// TwinCAT 3 PLC project TcSocketHelper_SingleServerBinary
// ProgramVersion: 3.1.0.5
// libraries:
//   Tc2_Standard, * (Beckhoff Automation GmbH)
//   Tc2_System, * (Beckhoff Automation GmbH)
//   Tc2_TcpIp, * (Beckhoff Automation GmbH)
//   Tc2_Utilities, * (Beckhoff Automation GmbH)
//   Tc3_Module, * (Beckhoff Automation GmbH)
// project tree:
//   Data types/ ST_ApplicationBinaryData.TcDUT, ST_BinaryFrame.TcDUT, ST_BinaryHeader.TcDUT
//   Global Variables/ Global_Variables.TcGVL
//   / PlcTaskServer.TcTTO
//   POUs/ FB_Server.TcPOU, FB_ServerApplication.TcPOU, FB_ServerConnection.TcPOU, MAIN.TcPOU
//   POUs/Helper POUs/ FB_FrameFifo.TcPOU (not stored), FB_LogFifo.TcPOU, F_ADSLOGHEXDATA.TcPOU
// real-time tasks:
//   TASK PlcTaskServer: cycle T#10ms, priority 21, ADS port 351

CONFIGURATION TcSocketHelper_SingleServerBinary
    RESOURCE PLC ON TwinCAT3
        TASK PlcTaskServer(INTERVAL := T#10ms, PRIORITY := 21);
        PROGRAM MAIN WITH PlcTaskServer : MAIN;
    END_RESOURCE
END_CONFIGURATION

// ---- Data types/ST_ApplicationBinaryData.TcDUT
(* Simple binary user data (8 byte aligned) *)
TYPE ST_ApplicationBinaryData :
STRUCT
	(* Adapt this structure to match your protocol needs *)
	
	dtTimeStamp : DT		:= DT#2008-12-01-00:00;(* 4 byte *)
	nVelo		: UDINT		:= 0;(* 4 byte *)
	fPos		: LREAL		:= 0.0;(* 8 byte *)
	arr	 		: ARRAY[0..19] OF BYTE;(* 20 byte *)

	sMsg		: STRING	:= 'None';(* 81 byte *)
	reserved	: ARRAY[0..2] OF BYTE;(* Alignment data: 3 byte *)

	(* Total user data size = 120 byte *)
END_STRUCT
END_TYPE

// ---- Data types/ST_BinaryFrame.TcDUT
(* Simple binary TCP/IP frame (8 byte aligned) *)
TYPE ST_BinaryFrame :
STRUCT
	head	: ST_BinaryHeader;(* Frame header (16 byte) *)
	data 	: ST_ApplicationBinaryData;(* User data (120 byte) *)

	(* Total frame size = 136 byte *)
END_STRUCT
END_TYPE

// ---- Data types/ST_BinaryHeader.TcDUT
(* Simple binary TCP/IP frame header (8 byte aligned) *)
TYPE ST_BinaryHeader :
STRUCT
	dwStart		: DWORD	:= 16#BECF1234;	(* Start bytes *)
	cbLength	: UDINT(0..PLCPRJ_BUFFER_SIZE) := 0;(* Max. length of attached binary data *)
	nS			: UDINT := 0;(* Send counter *)
	nR			: UDINT	:= 0;(* Receive counter *)
	
	(* Total header data size = 16 byte *)
END_STRUCT
END_TYPE

// ---- Global Variables/Global_Variables.TcGVL
VAR_GLOBAL CONSTANT
	PLCPRJ_BUFFER_SIZE						: UDINT := 1000;(* Max. internal fifo/receiver buffer size *)

(*	PLCPRJ_CLIENT_SEND_CYCLE_TIME			: TIME := T#1S; not used at server side *)
	PLCPRJ_RECEIVE_POLLING_TIME				: TIME := T#100MS;
	PLCPRJ_RECEIVE_TIMEOUT					: TIME := T#50S;

	(* Some project specific error codes *)
	PLCPRJ_ERROR_RECEIVE_TIMEOUT			: UDINT := 16#8101;(* Receive timeout *)
	PLCPRJ_ERROR_SENDFIFO_OVERFLOW			: UDINT := 16#8102;(* Send fifo overflow *)
	PLCPRJ_ERROR_RECFIFO_OVERFLOW			: UDINT := 16#8103;(* Receive fifo overflow *)
	PLCPRJ_ERROR_INVALID_FRAME_FORMAT		: UDINT := 16#8104;(* Invalid frame format/data *)
END_VAR

// ---- POUs/MAIN.TcPOU
PROGRAM MAIN
VAR
	sSrvNetID		: T_AmsNetID	:= '';(* TwinCAT TCP/IP server network address *)
	sLocalHost		: T_Ipv4Addr 	:= '127.0.0.1';(* Server IP network address *)
	nLocalPort		: UDINT 		:= 200;(* Server port number *)
	bEnable			: BOOL 			:= TRUE;(* TRUE => Enable server data exchange, FALSE => Disable *)
	bLog			: BOOL			:= TRUE;(* TRUE => Enable log message output, FALSE => Disable *)
	fbServer		: FB_Server := ( sPrefix := 'SERVER::' );(* Server (connection) instance *)
	hServer			: T_HSERVER;(* Server connection handle *)

	fbCloseAll		: FB_SocketCloseAll;
	bInitialize		: BOOL := TRUE;
END_VAR

(* On PLC reset or program download close all old (opened) connections *)
fbCloseAll( sSrvNetID := sSrvNetID, bExecute:= bInitialize );
IF fbCloseAll.bBusy OR fbCloseAll.bError THEN
	RETURN;
END_IF

IF bInitialize THEN
	bInitialize := FALSE;

	(* Initialize server handle *)
	F_CreateServerHnd( 	sSrvNetID 	:= sSrvNetID,
						sLocalHost 	:= sLocalHost,
						nLocalPort	:= nLocalPort,
						nMode 		:= SEL( bLog, 0, CONNECT_MODE_ENABLEDBG ),(* Enable debug messages *)
						bEnable 	:= FALSE,(* TRUE = leave listener socket open, FALSE = close listener socket after last connection ist closed too *)
						hServer 	:= hServer );
END_IF


(* Trigger the execution of every server (connection) instance *)
fbServer( hServer := hServer, sSrvNetID := sSrvNetID, bEnable := bEnable, bLog := bLog );

END_PROGRAM

// ---- POUs/FB_Server.TcPOU
FUNCTION_BLOCK FB_Server
VAR_IN_OUT
	hServer			: T_HSERVER;(* Server connection handle *)
END_VAR
VAR_INPUT
	sSrvNetID		: T_AmsNetID	:= '';(* TwinCAT TCP/IP server network address *)
	bEnable			: BOOL 			:= FALSE;(* TRUE => Enable server data exchange, FALSE => Disable *)
	bLog			: BOOL 			:= FALSE;(* TRUE => Enable log message output, FALSE => Disable *)
	sPrefix			: STRING 		:= 'SERVER::';(* Log message description string (allows the identification of log message source) *)
END_VAR
VAR_OUTPUT
	eState			: E_SocketConnectionState := eSOCKET_DISCONNECTED;(* TCP/IP connection state *)
END_VAR
VAR
	fbApplication 	: FB_ServerApplication;(* Server application control function block *)
	fbConnection	: FB_ServerConnection;(* Server data exchange control function block *)
	fbTx 			: FB_FrameFifo;(* Tx fifo *)
	fbRx 			: FB_FrameFifo;(* Rx fifo *)
	fbLog			: FB_LogFifo;(* Log/debug/error fifo *)
END_VAR

(*-------------------------- Trigger data exchange -----------------------------------------------*)
fbConnection( 	hServer := hServer, sSrvNetID := sSrvNetID, 
				fbRx := fbRx, fbTx := fbTx, fbLog := fbLog, 
				bEnable := bEnable, bLog := bLog, sPrefix := sPrefix, eState=>eState );
	
IF fbConnection.eState = eSOCKET_CONNECTED THEN(* Connection established *)
	fbApplication( fbTx := fbTx, fbRx := fbRx, fbLog := fbLog );
END_IF

END_FUNCTION_BLOCK

// ---- POUs/FB_ServerApplication.TcPOU
(* Sample server application. Adapt this code to match your needs. *)
FUNCTION_BLOCK FB_ServerApplication
VAR_IN_OUT
	fbTx 			: FB_FrameFifo;(* TX fifo *)
	fbRx 			: FB_FrameFifo;(* RX fifo *)
	fbLog			: FB_LogFifo;(* Log message fifo *)
END_VAR
VAR
	stToClient		: ST_ApplicationBinaryData; (* Tx user data *)
	stFromClient	: ST_ApplicationBinaryData; (* Rx user data *)
	sLogMessage 	: T_MaxString := '';(* Log/debug/error message *)
END_VAR

(*------------------- Fetch rx data and send them back to the client -------------------------------------------------- *)
REPEAT
	fbRx.RemoveHead( );(* Fetch data from rx fifo *)
	IF fbRx.bOk THEN(* Success *)

		stFromClient := fbRx.stGet;
		
		stToClient := stFromClient;
		stToClient.sMsg := 'Hello world from server!';(* Modify some of the client data *)
		

		(* Send data back to the client *)
		fbTx.AddTail( stPut := stToClient );(* Put user data to the tx fifo *)
		IF NOT fbTx.bOk THEN(* Fifo overflow => Log error *)
			fbLog.Error( sMessage := 'FB_FrameFifo(sender)', nErrID := PLCPRJ_ERROR_SENDFIFO_OVERFLOW );
		END_IF
	END_IF
UNTIL NOT fbRx.bOk
END_REPEAT

(*---------------------- Get log/error messages from log fifo ------------------*)
REPEAT
	fbLog.Remove( );
	IF fbLog.bOk THEN

		(* TODO: Implement log message handler *)
		sLogMessage := fbLog.sGet;

	END_IF
UNTIL NOT fbLog.bOk
END_REPEAT

END_FUNCTION_BLOCK

// ---- POUs/Helper POUs/FB_LogFifo.TcPOU
(* Log/debug/error message fifo *)
FUNCTION_BLOCK FB_LogFifo
VAR_INPUT
	bLog		: BOOL 		:= FALSE;(* TRUE => Enable log message output, FALSE => Disable *)
	sPrefix		: STRING 	:= 'Unknown::';(* Log message description string (allows the identification of log message source) *)
	
	sMessage	: STRING 	:= '';(* String message to add (write) to the fifo *)
	nErrID		: UDINT 	:= 0;(* Error code to add (write) to the fifo *)
	hSocket		: T_HSOCKET;(* Socket connection handle *)
END_VAR
VAR_OUTPUT
	bOk			: BOOL;(* TRUE = New entry added or removed succesfully, FALSE = Fifo overflow or fifo empty *)
	sGet		: T_MaxString := '';(* String entry removed (read) from fifo *)
	nCount		: UDINT := 0;(* Number of fifo entries *)
END_VAR
VAR
	fbBuffer 	: FB_StringRingBuffer;(* Basic (lower level) string buffer control function block *)
	buffer		: ARRAY[0..PLCPRJ_BUFFER_SIZE] OF BYTE;(* Internal buffer memory *)
	sSource		: T_MaxString;	
	sPut		: T_MaxString;
END_VAR

;

ACTION Error:
(* Adds new fifo entry *)
IF nErrID = 0 THEN
	sSource := '::Error: 0x';
ELSIF ( nErrID AND 16#80000000) = 16#80000000 THEN
	IF nErrID = 16#80072746 THEN
		sSource := '::Win32 error (the connection is reset by remote side): 0x';
	ELSE
		sSource := '::Win32 error: 0x';
	END_IF
ELSIF (nErrID AND 16#00008100) = 16#00008100 THEN
	CASE nErrID OF
		PLCPRJ_ERROR_RECEIVE_TIMEOUT:
			sSource := '::PLC sample project receive timeout error: 0x';
		PLCPRJ_ERROR_SENDFIFO_OVERFLOW:
			sSource := '::PLC sample project send fifo overflow error: 0x';
		PLCPRJ_ERROR_RECFIFO_OVERFLOW:
			sSource := '::PLC sample project receive fifo overflow error: 0x';
		PLCPRJ_ERROR_INVALID_FRAME_FORMAT:
			sSource := '::PLC sample project invalid frame format error: 0x';
	ELSE
		sSource := '::Other PLC sample project error: 0x';
	END_CASE
ELSIF (nErrID AND 16#00008000) = 16#00008000 THEN
	sSource := '::Internal TCP/IP Connection Server error: 0x';
ELSE
	sSource := '::TwinCAT System error: 0x';
END_IF

sPut := CONCAT( CONCAT( CONCAT( sPrefix, sMessage ), sSource ), DWORD_TO_HEXSTR( nErrID AND 16#FFFF, 0, FALSE ) ); 

fbBuffer.A_AddTail( pBuffer:= ADR(buffer), cbBuffer:= SIZEOF(buffer),
					putValue:= sPut, bOk=>bOk, nCount=>nCount );
IF bOk THEN
	IF bLog THEN(* Log error message *)
		ADSLOGSTR( ADSLOG_MSGTYPE_ERROR OR ADSLOG_MSGTYPE_LOG, '%s', sPut );	
	END_IF
END_IF
END_ACTION

ACTION Message:
(* Adds new fifo entry *)
sPut := CONCAT( CONCAT( sPrefix, sMessage ), CONCAT( '::', HSOCKET_TO_STRING(hSocket) ) );
fbBuffer.A_AddTail( pBuffer:= ADR(buffer), cbBuffer:= SIZEOF(buffer),
					putValue:= sPut, bOk=>bOk, nCount=>nCount );
IF bOk THEN
	IF bLog THEN(* Log information message *)
		ADSLOGSTR( ADSLOG_MSGTYPE_HINT OR ADSLOG_MSGTYPE_LOG, '%s', sPut );	
	END_IF
END_IF
END_ACTION

ACTION Remove:
(* Removes oldest fifo entry *)
IF nCount = 0 THEN
	sGet := '';
	bOk := FALSE;
	RETURN;
END_IF

fbBuffer.A_RemoveHead( pBuffer:= ADR(buffer), cbBuffer:= SIZEOF(buffer),
						getValue=>sGet, bOk=>bOk, nCount=>nCount );
END_ACTION

ACTION Clear:
(* Clears all fifo entries *)
fbBuffer.A_Reset( 	pBuffer := ADR( buffer ), cbBuffer := SIZEOF( buffer ), 
					bOk=>bOk, nCount=>nCount, getValue=>sGet );
END_ACTION

END_FUNCTION_BLOCK

// ---- POUs/FB_ServerConnection.TcPOU
(* 	This function block implements simple TCP/IP server protocol. *)
FUNCTION_BLOCK FB_ServerConnection
VAR_IN_OUT
	hServer		: T_HSERVER;(* Server connection handle *)
	fbTx 		: FB_FrameFifo;(* TX fifo *)
	fbRx 		: FB_FrameFifo;(* RX fifo *)
	fbLog		: FB_LogFifo;(* Log message fifo *)
END_VAR
VAR_INPUT
	sSrvNetID	: T_AmsNetID	:= '';(* TwinCAT TCP/IP server network address *)
	bEnable		: BOOL			:= FALSE;(* TRUE => Enable/connect, FALSE => Disable/disconnect *)
	tReconnect	: TIME 			:= T#1S;(* Try to reconnect after this time *)
	bLog		: BOOL 			:= FALSE; (* TRUE => Enable debug output, FALSE => Disable debug output *)
	sPrefix		: STRING 		:= 'SERVER::';(* Log message description string (allows the identification of log message source) *)
END_VAR
VAR_OUTPUT
	eState		: E_SocketConnectionState := eSOCKET_DISCONNECTED;(* TCP/IP connection state *)
END_VAR
VAR
	fbConnect 	: FB_ServerClientConnection;(* Create/release TCP/IP connection *)
	fbSend		: FB_SocketSend;(* Send TCP/IP data *)
	fbReceive	: FB_SocketReceive;(* Receive TCP/IP data *)
	nState 		: BYTE;(* Global state *)
	bSndBusy 	: BOOL;(* Tx state *)
	bRcvBusy 	: BOOL;(* Rx state *)
	bDisconnect	: BOOL;(* Disconnect flag, if set the socket will be closed *)

	fbPollTimer	: TON;(* Rx data poll timer *)
	fbRequestTimer	: TON;(* Request timeout timer *)
	fbReconnectTimer : TON;(* Reconnect timer *)

	nS			: UDINT;(* Send frame counter *)
	nR			: UDINT;(* Received frame counter *)
	cbReceived	: UDINT;(* Count of received data bytes *)
	rxBuffer	: ARRAY[0..PLCPRJ_BUFFER_SIZE] OF BYTE;
	cbFrame		: UDINT;(* Rx frame byte size *)
	stTxFrame	: ST_BinaryFrame;(* Tx frame buffer (inclusive header) *)
	stRxFrame	: ST_BinaryFrame;(* Rx frame buffer (inclusive header) *)
	bAbort		: BOOL;(* Flag to abort frame parsing loop *)
END_VAR

CASE nState OF
	0:(* Create TCP/IP connection *)
		fbConnect( 	eMode := eACCEPT_ALL, tReconnect := tReconnect, bEnable := bEnable, 
					hServer := hServer, eState => eState );
		IF NOT fbConnect.bBusy THEN
			IF NOT fbConnect.bError THEN
				IF eState = eSOCKET_CONNECTED THEN(* we are connected *)
					
					fbTx.Clear( sPrefix := CONCAT( sPrefix, 'FB_FrameFifo(sender)::' ), bLog := bLog );(* Clear TX fifo (optional) *)
					fbRx.Clear( sPrefix := CONCAT( sPrefix, 'FB_FrameFifo(receiver)::' ), bLog := bLog );(* Clear RX fifo (optional) *)
					fbLog.Clear( sPrefix := sPrefix, bLog := bLog );(* Clear log fifo (optional) *)
					bSndBusy := FALSE;
					bRcvBusy := FALSE;
					bDisconnect := FALSE;
					cbReceived 	:= 0;(* Reset number of received data bytes *)
					nR 			:= 0;(* Reset receive frame counter *)
					nS 			:= 0;(* Reset send frame counter *)

					fbPollTimer( IN := FALSE, PT := T#0S );
					fbRequestTimer( IN := FALSE, PT := PLCPRJ_RECEIVE_TIMEOUT );
					fbReconnectTimer( IN := FALSE, PT := tReconnect );
				
					fbLog.Message( sMessage := 'Connection established!', hSocket := fbConnect.hSocket );
					nState 	:= 1;
				END_IF
			ELSE(* Connect error => log error *)
				fbLog.Error( sMessage := 'FB_ServerClientConnection()', nErrID := fbConnect.nErrId );
			END_IF
		END_IF


	1:(* Data exchange state *)
		bDisconnect := NOT bEnable OR bDisconnect;(* User/internal disconnect requested? *)
		IF bDisconnect AND NOT bSndBusy AND NOT bRcvBusy THEN
			bDisconnect := FALSE;
			fbLog.Message( sMessage := 'Closing connection!', hSocket := fbConnect.hSocket );
			nState := 2;(* Disconnect *)
		ELSE

			(* ----------------------- Get/fetch rx data -------------------------------- *)
			IF NOT bDisconnect AND NOT bRcvBusy THEN
				fbPollTimer( IN := TRUE );
				IF fbPollTimer.Q THEN
					IF fbRx.cbFree >= SIZEOF(stRxFrame.data) THEN(* Check free rx fifo space *)
						fbPollTimer( IN := FALSE, PT := PLCPRJ_RECEIVE_POLLING_TIME );
						fbReceive( bExecute := FALSE );
						fbReceive( 	sSrvNetId	:= sSrvNetID,
									hSocket		:= fbConnect.hSocket,
									cbLen		:= SIZEOF(rxBuffer) - cbReceived,
									pDest		:= ADR(rxBuffer) + cbReceived,
									bExecute	:= TRUE );
						bRcvBusy := TRUE;
					END_IF
				END_IF
				
			ELSE(* Wait until receive not busy *)
				
				fbReceive( bExecute := FALSE );
				IF NOT fbReceive.bBusy THEN
					bRcvBusy := FALSE;
					IF NOT fbReceive.bError THEN
						IF fbReceive.nRecBytes > 0 THEN (* Some bytes received *)

							fbPollTimer( IN := FALSE, PT := T#0S );(* Bytes received => increase the read (polling) speed *)
							fbRequestTimer( IN := FALSE );(* Bytes received => disable timeout check *)
							cbReceived := cbReceived + fbReceive.nRecBytes;

							(* Parse received bytes *)
							REPEAT
								bAbort := TRUE;(* Set flag *)
								
								IF cbReceived >= SIZEOF(stRxFrame.head) THEN (* All header bytes received => check header data *)
									
									MEMCPY( ADR( stRxFrame.head ), ADR( rxBuffer ), SIZEOF( stRxFrame.head ) );(* Get header data *)
								
									IF (stRxFrame.head.dwStart = 16#BECF1234) (* Check start bytes *)
									AND (stRxFrame.head.nS = nR )(* Check counter (send counter == expected receive counter?) *)
									AND (stRxFrame.head.cbLength <= SIZEOF(stRxFrame.data))(* Check frame (user data) length *)
									THEN
									
										cbFrame := SIZEOF(stRxFrame.head) + stRxFrame.head.cbLength;(* Calculate the expected receive frame length *)
										IF cbReceived >= cbFrame  THEN (* All frame (user data) bytes received? *)
	
											MEMCPY( ADR( stRxFrame ), ADR( rxBuffer ), MIN( SIZEOF(stRxFrame), cbFrame ) );
											fbRx.AddTail( stPut := stRxFrame.data );(* Add user data to the rx fifo *)
											IF fbRx.bOk THEN
												nR := nR + 1;(* Increment receive counter *)

												MEMMOVE( ADR( rxBuffer ), ADR( rxBuffer ) + cbFrame, cbReceived - cbFrame );(* Shift the remaining rx bytes *)
												cbReceived := cbReceived - cbFrame;(* Recalculate the size of the remaining rx bytes *)

												IF fbRx.cbFree >= SIZEOF(stRxFrame.data) THEN
													bAbort := FALSE;(* reset flag, try to parse next frame *)
												END_IF
											ELSE (* Fifo overflow => log error and disconnect *)
												fbLog.Error( sMessage := 'FB_FrameFifo(receiver)', nErrID := PLCPRJ_ERROR_RECFIFO_OVERFLOW );
												bDisconnect := TRUE;(* Set flag *)
												RETURN;
											END_IF

(*										ELSE repeat reading *)
										END_IF

									ELSE(* Receive error => Invalid frame format/data *)
										fbLog.Error( sMessage := 'FB_ServerConnection()', nErrID := PLCPRJ_ERROR_INVALID_FRAME_FORMAT );
										bDisconnect := TRUE;(* Set flag *)
										RETURN;
									END_IF

(*								ELSE repeat reading *)
								END_IF (* IF cbReceived >= SIZEOF(stRxFrame.head) THEN *)

							UNTIL bAbort
							END_REPEAT

						ELSE(* No bytes received *)
							fbRequestTimer( IN := TRUE );(* No bytes received => enable timeout check *)
							IF fbRequestTimer.Q THEN (* Timeout error*)
								fbRequestTimer( IN := FALSE );
								fbLog.Error( sMessage := 'FB_ServerConnection()', nErrID := PLCPRJ_ERROR_RECEIVE_TIMEOUT );
								bDisconnect := TRUE;(* Set flag *)
							END_IF							
						END_IF(* IF fbReceive.nRecBytes > 0 THEN *)

					ELSE(* Receive error => Log error and disconnect *)
						fbLog.Error( sMessage := 'FB_SocketReceive()', nErrID := fbReceive.nErrId );
						bDisconnect := TRUE;(* set flag *)
					END_IF

				END_IF(* IF NOT fbReceive.bBusy THEN *)
				
			END_IF(* IF NOT bDisconnect AND NOT bRcvBusy THEN *)
			(* -------------------------------------------------------------------------- *)

			
			
			(* ------------------------------ Send tx data ------------------------------ *)
			IF NOT bDisconnect AND NOT bSndBusy THEN
				fbTx.RemoveHead();(* Remove oldest user data entry *)
				IF fbTx.bOk THEN(* Success *)
						
					stTxFrame.data := fbTx.stGet;
					
					(* Append/create some protocol header *)
					stTxFrame.head.dwStart 	:= 16#BECF1234;(* Frame start bytes *)
					stTxFrame.head.cbLength := SIZEOF( stTxFrame.data);(* Set length of user data *)
					stTxFrame.head.nS 		:= nS;(* Number of send frames *)
					stTxFrame.head.nR 		:= nR;(* Number of received frames *)
					
					(* Send frame *)
					fbSend( bExecute := FALSE );
					fbSend(	sSrvNetID 	:= sSrvNetID,
							hSocket		:= fbConnect.hSocket,
							cbLen		:= SIZEOF(stTxFrame),(* Size of header + size of user data *)
							pSrc		:= ADR(stTxFrame),(* Pointer to the frame data *)
							bExecute	:= TRUE );
					bSndBusy := TRUE;
				END_IF
			ELSE(* Wait until send not busy *)
				fbSend( bExecute := FALSE );
				IF NOT fbSend.bBusy THEN
					bSndBusy := FALSE;
					IF NOT fbSend.bError THEN(* No error *)
						nS := nS + 1;(* Increment the number of send frames *)
					ELSE(* Send error => Log error and disconnect *)
						fbLog.Error( sMessage := 'FB_SocketSend()', nErrID := fbSend.nErrId );
						bDisconnect := TRUE;(* Set flag *)
					END_IF
				END_IF
			END_IF
			(* -------------------------------------------------------------------------- *)

			
		END_IF(* IF bDisconnect AND NOT bSndBusy AND NOT bRcvBusy THEN *)


	2:(* Disconnect *)
		fbConnect( hServer := hServer, bEnable:= FALSE, eState=>eState );
		IF eState = eSOCKET_DISCONNECTED THEN
			fbReconnectTimer( IN := TRUE );(* Please wait some seconds and then try to connect again *)
			IF fbReconnectTimer.Q THEN
				fbReconnectTimer( IN := FALSE );
				nState := 0;
			END_IF
		END_IF

END_CASE

END_FUNCTION_BLOCK

// ---- POUs/Helper POUs/F_ADSLOGHEXDATA.TcPOU
(* This function logs hexadecimal data to the TwinCAT XAE->Error list window *)
FUNCTION F_ADSLOGHEXDATA : DINT
VAR_INPUT
	sPrefix		: STRING;(* Debug message prefix string (allows the identification of log message source) *)
	pBuffer		: PVOID;(* Address of source buffer *)
	cbBuffer	: UDINT;(* Byte size of source buffer *)
END_VAR
VAR
	fbSplit	: FB_MemBufferSplit;
	sArg	: T_MaxString;
	sFormat : STRING;
END_VAR

IF pBuffer = 0 OR cbBuffer = 0 THEN
	RETURN;
END_IF

sFormat := CONCAT( sPrefix, '%s' );
fbSplit.eCmd := eEnumCmd_First;

REPEAT
	fbSplit( pBuffer := pBuffer, cbBuffer := cbBuffer, cbSize := 32 );(* Split binary data to 32 byte segments *)
	IF fbSplit.bOk THEN

		sArg := DATA_TO_HEXSTR( pData := fbSplit.pSegment, cbData := fbSplit.cbSegment, FALSE );(* Convert binary data to hex string *)

		F_ADSLOGHEXDATA := ADSLOGSTR( ADSLOG_MSGTYPE_HINT OR ADSLOG_MSGTYPE_LOG, sFormat, sArg );(* Log hex string *)

		sFormat := '%s';
		fbSplit.eCmd := eEnumCmd_Next;
	END_IF
UNTIL NOT fbSplit.bOk
END_REPEAT

END_FUNCTION
